// TIA Portal V17 export
// export: Created 2023-02-26T22:59:49.6061549Z, ExportSetting WithDefaults, DisplayName Totally Integrated Automation Portal, DisplayVersion V17, DisplayName TIA Portal Openness, DisplayVersion V17, DisplayName TIA Portal Version Control Interface, DisplayVersion V17, DisplayName TIA Portal Test Suite Advanced, DisplayVersion V17, DisplayName STEP 7 Professional, DisplayVersion V17, DisplayName SIMATIC Energy Suite, DisplayVersion V17, DisplayName STEP 7 Safety, DisplayVersion V17, DisplayName WinCC Professional, DisplayVersion V17
FUNCTION "LOG_Statistic" : Void   // FC8, LAD
{ S7_Optimized_Access := 'TRUE' }
VERSION : 0.1
// stored: AutoNumber false, IsIECCheckEnabled false, SetENOAutomatically false, UDAEnableTagReadback false
   VAR_TEMP
      t_RisingEdge : Bool;
   END_VAR
BEGIN

REGION Network 1: Call: CountPackages
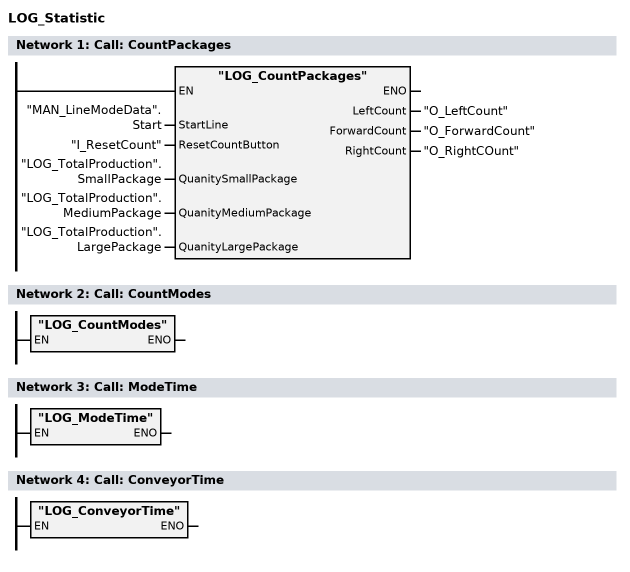
   RUNG wire#powerrail
      "LOG_CountPackages"(StartLine := "MAN_LineModeData".Start, ResetCountButton := "I_ResetCount", QuanitySmallPackage := "LOG_TotalProduction".SmallPackage, QuanityMediumPackage := "LOG_TotalProduction".MediumPackage, QuanityLargePackage := "LOG_TotalProduction".LargePackage, LeftCount => "O_LeftCount", ForwardCount => "O_ForwardCount", RightCount => "O_RightCOunt")
   END_RUNG
   // the same network as SCL:
   "LOG_CountPackages"(StartLine := "MAN_LineModeData".Start,
                       ResetCountButton := "I_ResetCount",
                       QuanitySmallPackage := "LOG_TotalProduction".SmallPackage,
                       QuanityMediumPackage := "LOG_TotalProduction".MediumPackage,
                       QuanityLargePackage := "LOG_TotalProduction".LargePackage,
                       LeftCount => "O_LeftCount",
                       ForwardCount => "O_ForwardCount",
                       RightCount => "O_RightCOunt");
END_REGION

REGION Network 2: Call: CountModes
   RUNG wire#powerrail
      "LOG_CountModes"()
   END_RUNG
   // the same network as SCL:
   "LOG_CountModes"();
END_REGION

REGION Network 3: Call: ModeTime
   RUNG wire#powerrail
      "LOG_ModeTime"()
   END_RUNG
   // the same network as SCL:
   "LOG_ModeTime"();
END_REGION

REGION Network 4: Call: ConveyorTime
   RUNG wire#powerrail
      "LOG_ConveyorTime"()
   END_RUNG
   // the same network as SCL:
   "LOG_ConveyorTime"();
END_REGION
END_FUNCTION
